PROGRAM MAPPING_out
VAR CONSTANT
{IF defined (AXIS_MAP)}
  {info 'MAPPING_out - ACTIVE'}
  bBypassMapping    : BOOL  := FALSE;
{ELSE}
  bBypassMapping    : BOOL  := TRUE;
{END_IF}
END_VAR
VAR
  AxisState         : U_AXIS_STATE;
  AxisInfo          : U_AXIS_INFO;
  AxisParameterRd   : U_AXIS_NC_PARAMETER;

  nAxis             : INT;
END_VAR

IF bBypassMapping THEN RETURN; END_IF

FOR nAxis := 1 TO GVL_AXIS_CTRL.gciMaxAxis
DO
  AxisState.stState[nAxis]        := GVL_AXIS_CTRL.gstAxisControl[nAxis].FromPlc;
  AxisInfo.stState[nAxis]         := GVL_AXIS_CTRL.gfbAxisController[nAxis].StatusCompact;

  AxisParameterRd.stState[nAxis]  := GVL_AXIS_CTRL.gstAxisParam[nAxis];
END_FOR

END_PROGRAM

(* stored: Version 1.1.0.1, ProductVersion 3.1.4024.12
   POU MAPPING_out: Id {2f982087-90b2-048b-1461-b5f12ca1e4da}, SpecialFunc None *)
